Fanuc KAREL source: IO0093.KL

-- PROVISIONAL review KL for V1013-1; original PC SHA256 952db82c5c17072ff70c51022200d9c9e568db601f704a43c6faece254a927df
-- Incomplete behavior may be omitted. Consult companion uncertainty JSON. Do not deploy.
PROGRAM IO0093
%NOLOCKGROUP
-- UNRESOLVED_LOCAL_POOL 5 cells at code offset 13; source declarations unknown
-- DIRECT_LOCAL_WORD_ACCESS alone does not prove INTEGER, REAL, or BOOLEAN
BEGIN
  -- UNRESOLVED_PC offsets 0-18; opcodes 2B,2C,7B
  -- UNRESOLVED_PC offsets 23-30; opcodes 9D,23
  -- UNRESOLVED_PC offsets 35-49; opcodes 2E,22,9D,33,35
  -- UNRESOLVED_PC offsets 54-61; opcodes 9D,23
  -- UNRESOLVED_PC offsets 66-77; opcodes 2E,23
  -- UNRESOLVED_PC offsets 82-105; opcodes 22,21,33,34,19,9C,5B,79
  -- UNRESOLVED_PC offsets 110-124; opcodes 21,9D,52,23
  -- UNRESOLVED_PC offsets 134-138; opcodes 7F
  -- UNRESOLVED_PC offsets 143-147; opcodes 27,AA
  -- UNRESOLVED_PC offsets 152-156; opcodes 7F
END IO0093
